{attribute 'qualified_only'}
{attribute 'strict'}
TYPE E_EasyTempState :
(
	Stopped := 0,
	Running := 1,
	Tuning := 2,
	Resetting := 99
);
END_TYPE

(* stored: Version 1.1.0.1, ProductVersion 3.1.4024.12
   DUT E_EasyTempState: Id {a8dbd2af-b069-47e6-976c-e452f603a998} *)
